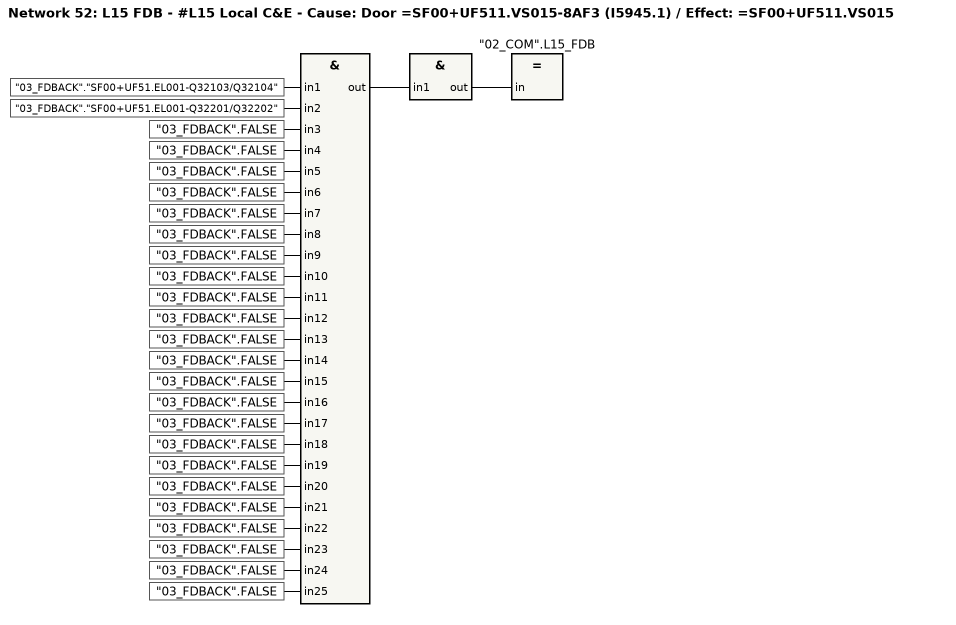
   "02_COM".L15_FDB := "03_FDBACK"."SF00+UF51.EL001-Q32103/Q32104" AND "03_FDBACK"."SF00+UF51.EL001-Q32201/Q32202" AND "03_FDBACK".FALSE AND "03_FDBACK".FALSE AND "03_FDBACK".FALSE AND "03_FDBACK".FALSE AND "03_FDBACK".FALSE AND "03_FDBACK".FALSE AND "03_FDBACK".FALSE AND "03_FDBACK".FALSE AND "03_FDBACK".FALSE AND "03_FDBACK".FALSE AND "03_FDBACK".FALSE AND "03_FDBACK".FALSE AND "03_FDBACK".FALSE AND "03_FDBACK".FALSE AND "03_FDBACK".FALSE AND "03_FDBACK".FALSE AND "03_FDBACK".FALSE AND "03_FDBACK".FALSE AND "03_FDBACK".FALSE AND "03_FDBACK".FALSE AND "03_FDBACK".FALSE AND "03_FDBACK".FALSE AND "03_FDBACK".FALSE;
END_REGION
END_FUNCTION
